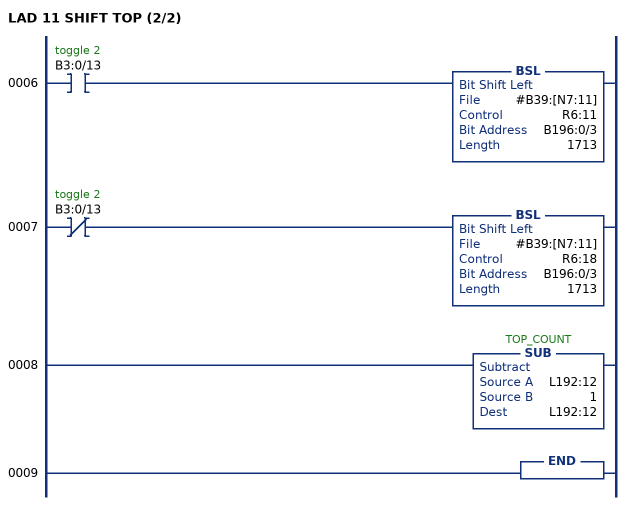
% Rung: 6 %
SOR XIC B3:0/13 BSL #B39:[N7:11] R6:11 B196:0/3 1713 EOR
%   B3:0/13  "toggle 2" %
%   N7:11  TOP_GOOD2_START_WORD %
%   B196:0/3  OFF %
% Rung: 7 %
SOR XIO B3:0/13 BSL #B39:[N7:11] R6:18 B196:0/3 1713 EOR
%   B3:0/13  "toggle 2" %
%   N7:11  TOP_GOOD2_START_WORD %
%   B196:0/3  OFF %
% Rung: 8 %
SOR SUB L192:12 1 L192:12 EOR
%   L192:12  TOP_COUNT %
% Rung: 9 %
SOR END EOR

LADDER 12 "BOTOPTIC"
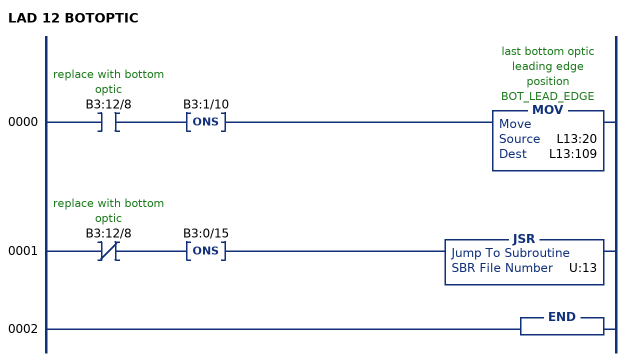
% Rung: 0 %
SOR XIC B3:12/8 ONS B3:1/10 MOV L13:20 L13:109 EOR
%   B3:12/8  "replace with bottom optic" %
%   L13:20  BOT_POSITION %
%   L13:109  BOT_LEAD_EDGE  "last bottom optic leading edge position" %
% Rung: 1 %
SOR XIO B3:12/8 ONS B3:0/15 JSR U:13 EOR
%   B3:12/8  "replace with bottom optic" %
% Rung: 2 %
SOR END EOR

LADDER 13 "BOTOPTMES"
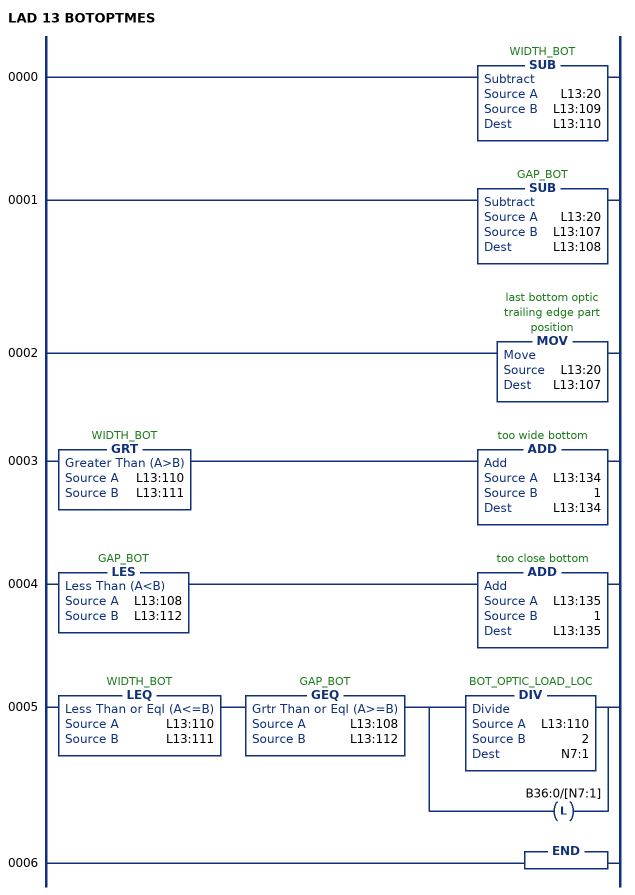
% Rung: 0 %
SOR SUB L13:20 L13:109 L13:110 EOR
%   L13:20  BOT_POSITION %
%   L13:109  BOT_LEAD_EDGE  "last bottom optic leading edge position" %
%   L13:110  WIDTH_BOT %
% Rung: 1 %
SOR SUB L13:20 L13:107 L13:108 EOR
%   L13:20  BOT_POSITION %
%   L13:107  "last bottom optic trailing edge part position" %
%   L13:108  GAP_BOT %
% Rung: 2 %
SOR MOV L13:20 L13:107 EOR
%   L13:20  BOT_POSITION %
%   L13:107  "last bottom optic trailing edge part position" %
% Rung: 3 %
SOR GRT L13:110 L13:111 ADD L13:134 1 L13:134 EOR
%   L13:110  WIDTH_BOT %
%   L13:111  BOT_MAX_WIDTH %
%   L13:134  "too wide bottom" %
% Rung: 4 %
SOR LES L13:108 L13:112 ADD L13:135 1 L13:135 EOR
%   L13:108  GAP_BOT %
%   L13:112  BOT_MIN_GAP %
%   L13:135  "too close bottom" %
% Rung: 5 %
SOR LEQ L13:110 L13:111 GEQ L13:108 L13:112 BST DIV L13:110 2 N7:1 NXB OTL B36:0/[N7:1] BND EOR
%   L13:110  WIDTH_BOT %
%   L13:111  BOT_MAX_WIDTH %
%   L13:108  GAP_BOT %
%   L13:112  BOT_MIN_GAP %
%   N7:1  BOT_OPTIC_LOAD_LOC %
%   B36:0  BOT_GOOD %
% Rung: 6 %
SOR END EOR

LADDER 135 "XFER"
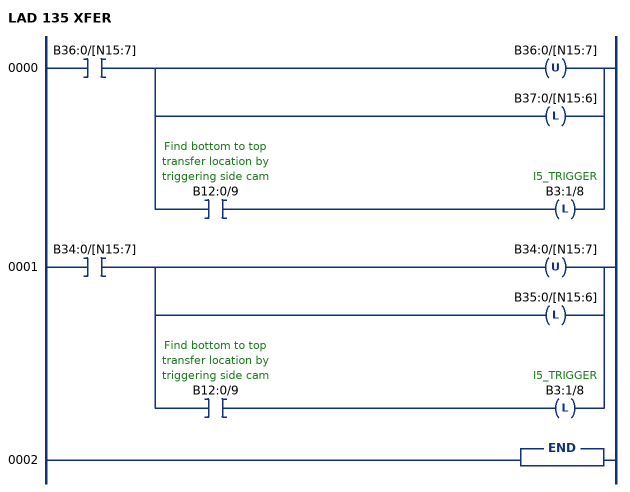
% Rung: 0 %
SOR XIC B36:0/[N15:7] BST OTU B36:0/[N15:7] NXB OTL B37:0/[N15:6] NXB XIC B12:0/9 OTL B3:1/8 BND EOR
%   B36:0  BOT_GOOD %
%   N15:7  XFER_OUT_LOC %
%   B37:0  TOPGOOD1 %
%   N15:6  XFER_IN_LOC %
%   B12:0/9  "Find bottom to top transfer location by triggering side cam" %
%   B3:1/8  I5_TRIGGER %
% Rung: 1 %
SOR XIC B34:0/[N15:7] BST OTU B34:0/[N15:7] NXB OTL B35:0/[N15:6] NXB XIC B12:0/9 OTL B3:1/8 BND EOR
%   B34:0  BOT_NG %
%   N15:7  XFER_OUT_LOC %
%   B35:0  TOP_NG %
%   N15:6  XFER_IN_LOC %
%   B12:0/9  "Find bottom to top transfer location by triggering side cam" %
%   B3:1/8  I5_TRIGGER %
% Rung: 2 %
SOR END EOR

LADDER 137 "TOPOPTIC"
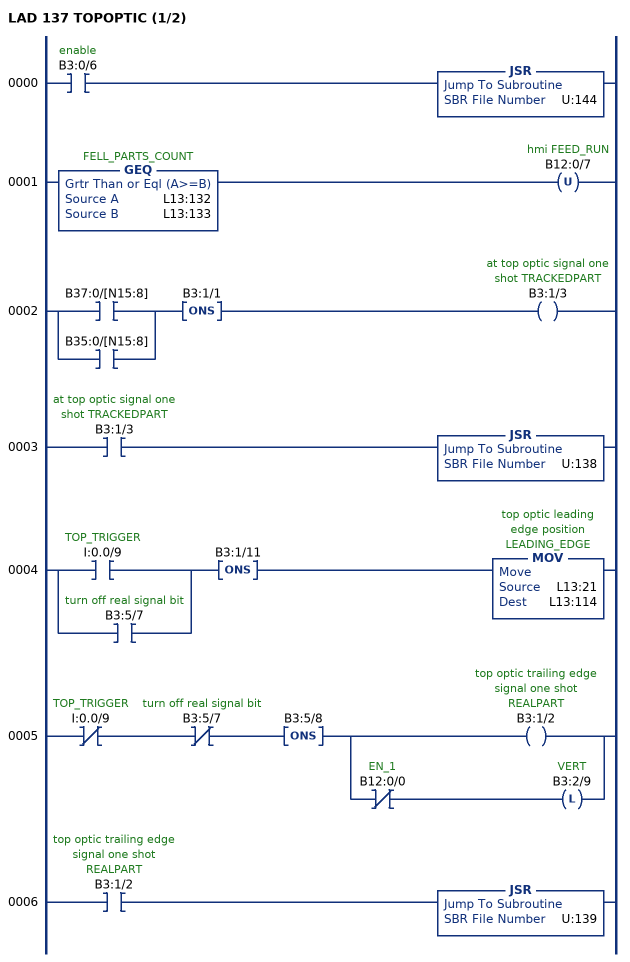
% Rung: 0 %
SOR XIC B3:0/6 JSR U:144 EOR
%   B3:0/6  "enable" %
% Rung: 1 %
SOR GEQ L13:132 L13:133 OTU B12:0/7 EOR
%   L13:132  FELL_PARTS_COUNT %
%   L13:133  FELL_PARTS_LIMIT %
%   B12:0/7  FEED_RUN  "hmi" %
% Rung: 2 %
SOR BST XIC B37:0/[N15:8] NXB XIC B35:0/[N15:8] BND ONS B3:1/1 OTE B3:1/3 EOR
%   B37:0  TOPGOOD1 %
%   N15:8  TOP_OPTIC_LOC %
%   B35:0  TOP_NG %
%   B3:1/3  TRACKEDPART  "at top optic signal one shot" %
% Rung: 3 %
SOR XIC B3:1/3 JSR U:138 EOR
%   B3:1/3  TRACKEDPART  "at top optic signal one shot" %
% Rung: 4 %
SOR BST XIC I:0.0/9 NXB XIC B3:5/7 BND ONS B3:1/11 MOV L13:21 L13:114 EOR
%   I:0.0/9  TOP_TRIGGER %
%   B3:5/7  "turn off real signal bit" %
%   L13:21  TOP_POSITION %
%   L13:114  LEADING_EDGE  "top optic leading edge position" %
% Rung: 5 %
SOR XIO I:0.0/9 XIO B3:5/7 ONS B3:5/8 BST OTE B3:1/2 NXB XIO B12:0/0 OTL B3:2/9 BND EOR
%   I:0.0/9  TOP_TRIGGER %
%   B3:5/7  "turn off real signal bit" %
%   B3:1/2  REALPART  "top optic trailing edge signal one shot" %
%   B12:0/0  EN_1 %
%   B3:2/9  VERT %
% Rung: 6 %
SOR XIC B3:1/2 JSR U:139 EOR
%   B3:1/2  REALPART  "top optic trailing edge signal one shot" %

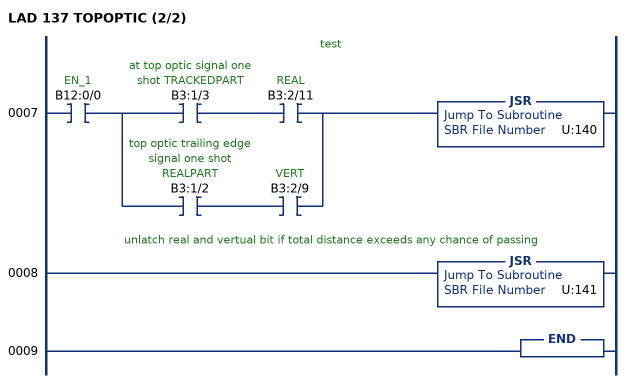
% Rung: 7 %
% test %
SOR XIC B12:0/0 BST XIC B3:1/3 XIC B3:2/11 NXB XIC B3:1/2 XIC B3:2/9 BND JSR U:140 EOR
%   B12:0/0  EN_1 %
%   B3:1/3  TRACKEDPART  "at top optic signal one shot" %
%   B3:2/11  REAL %
%   B3:1/2  REALPART  "top optic trailing edge signal one shot" %
%   B3:2/9  VERT %
% Rung: 8 %
% unlatch real and vertual bit if total distance exceeds any chance of passing %
SOR JSR U:141 EOR
% Rung: 9 %
SOR END EOR

LADDER 138 "TOPOPVERT"
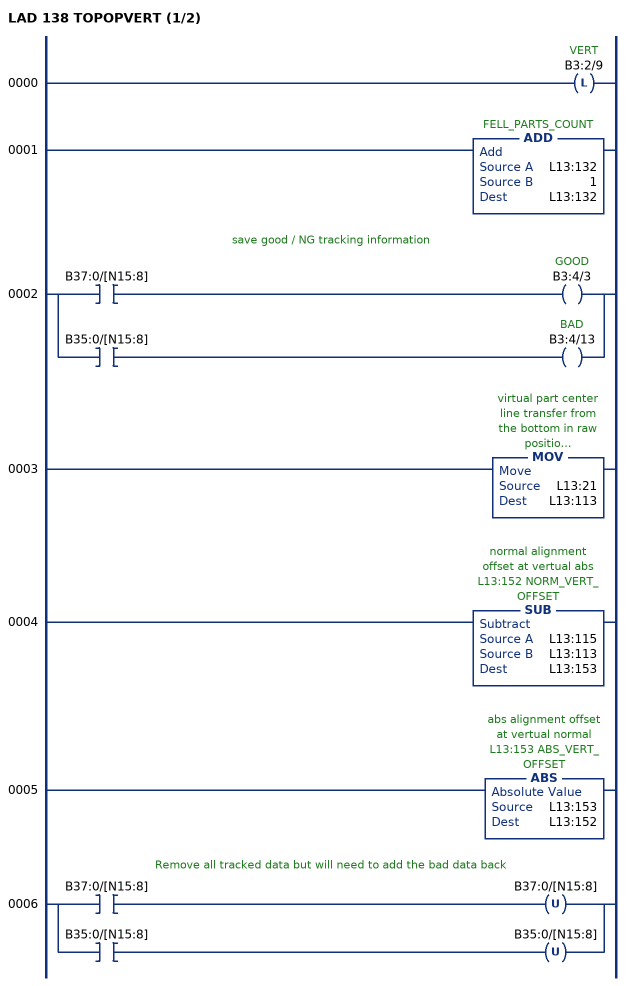
% Rung: 0 %
SOR OTL B3:2/9 EOR
%   B3:2/9  VERT %
% Rung: 1 %
SOR ADD L13:132 1 L13:132 EOR
%   L13:132  FELL_PARTS_COUNT %
% Rung: 2 %
% save good / NG tracking information %
SOR BST XIC B37:0/[N15:8] OTE B3:4/3 NXB XIC B35:0/[N15:8] OTE B3:4/13 BND EOR
%   B37:0  TOPGOOD1 %
%   N15:8  TOP_OPTIC_LOC %
%   B3:4/3  GOOD %
%   B35:0  TOP_NG %
%   B3:4/13  BAD %
% Rung: 3 %
SOR MOV L13:21 L13:113 EOR
%   L13:21  TOP_POSITION %
%   L13:113  VERTUAL_PT_RAW_CL  "virtual part center line transfer from the bottom in raw position" %
% Rung: 4 %
SOR SUB L13:115 L13:113 L13:153 EOR
%   L13:115  TRAILING_EDGE_RAW  "top optic trailing edge position" %
%   L13:113  VERTUAL_PT_RAW_CL  "virtual part center line transfer from the bottom in raw position" %
%   L13:153  NORM_VERT_OFFSET  "normal alignment offset at vertual abs L13:152" %
% Rung: 5 %
SOR ABS L13:153 L13:152 EOR
%   L13:153  NORM_VERT_OFFSET  "normal alignment offset at vertual abs L13:152" %
%   L13:152  ABS_VERT_OFFSET  "abs alignment offset at vertual normal L13:153" %
% Rung: 6 %
% Remove all tracked data but will need to add the bad data back %
SOR BST XIC B37:0/[N15:8] OTU B37:0/[N15:8] NXB XIC B35:0/[N15:8] OTU B35:0/[N15:8] BND EOR
%   B37:0  TOPGOOD1 %
%   N15:8  TOP_OPTIC_LOC %
%   B35:0  TOP_NG %

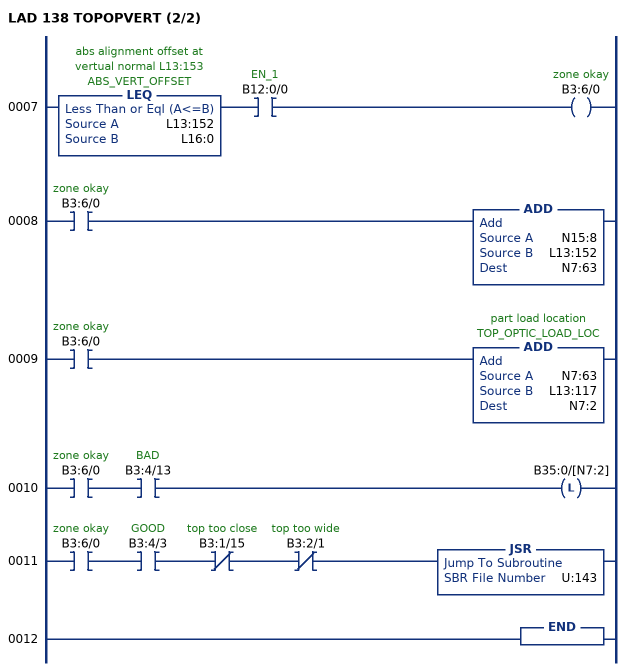
% Rung: 7 %
SOR LEQ L13:152 L16:0 XIC B12:0/0 OTE B3:6/0 EOR
%   L13:152  ABS_VERT_OFFSET  "abs alignment offset at vertual normal L13:153" %
%   L16:0  MAX_OFFSET %
%   B12:0/0  EN_1 %
%   B3:6/0  "zone okay" %
% Rung: 8 %
SOR XIC B3:6/0 ADD N15:8 L13:152 N7:63 EOR
%   B3:6/0  "zone okay" %
%   N15:8  TOP_OPTIC_LOC %
%   L13:152  ABS_VERT_OFFSET  "abs alignment offset at vertual normal L13:153" %
% Rung: 9 %
SOR XIC B3:6/0 ADD N7:63 L13:117 N7:2 EOR
%   B3:6/0  "zone okay" %
%   L13:117  HALF_WIDTH  "1/2 width top" %
%   N7:2  TOP_OPTIC_LOAD_LOC  "part load location" %
% Rung: 10 %
SOR XIC B3:6/0 XIC B3:4/13 OTL B35:0/[N7:2] EOR
%   B3:6/0  "zone okay" %
%   B3:4/13  BAD %
%   B35:0  TOP_NG %
%   N7:2  TOP_OPTIC_LOAD_LOC  "part load location" %
% Rung: 11 %
SOR XIC B3:6/0 XIC B3:4/3 XIO B3:1/15 XIO B3:2/1 JSR U:143 EOR
%   B3:6/0  "zone okay" %
%   B3:4/3  GOOD %
%   B3:1/15  "top too close" %
%   B3:2/1  "top too wide" %
% Rung: 12 %
SOR END EOR

LADDER 139 "TOPOPREAL"
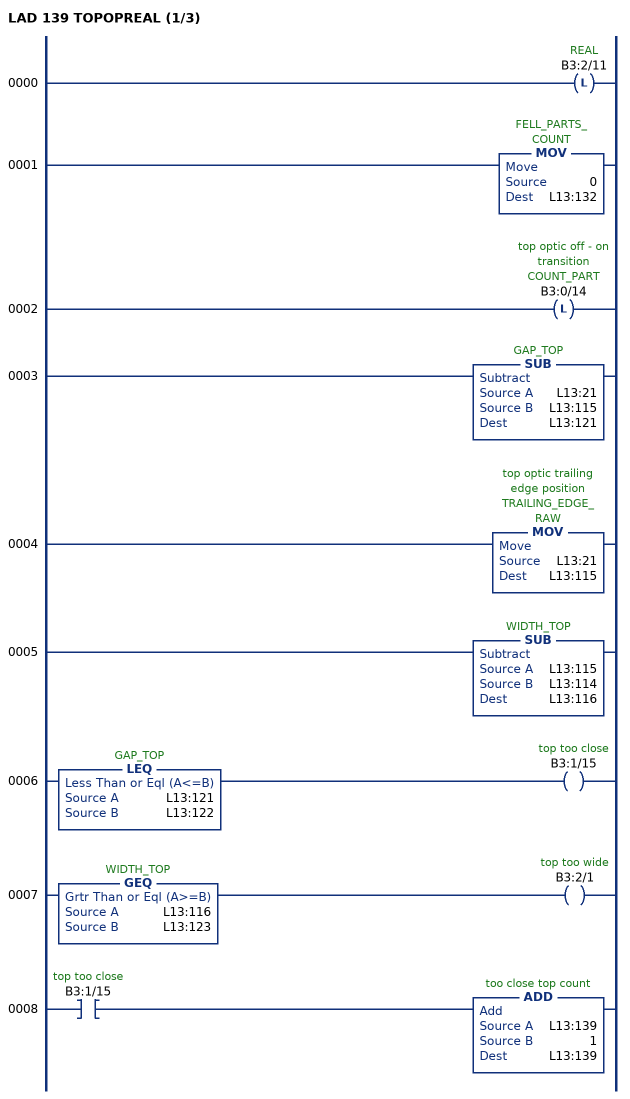
% Rung: 0 %
SOR OTL B3:2/11 EOR
%   B3:2/11  REAL %
% Rung: 1 %
SOR MOV 0 L13:132 EOR
%   L13:132  FELL_PARTS_COUNT %
% Rung: 2 %
SOR OTL B3:0/14 EOR
%   B3:0/14  COUNT_PART  "top optic off - on transition" %
% Rung: 3 %
SOR SUB L13:21 L13:115 L13:121 EOR
%   L13:21  TOP_POSITION %
%   L13:115  TRAILING_EDGE_RAW  "top optic trailing edge position" %
%   L13:121  GAP_TOP %
% Rung: 4 %
SOR MOV L13:21 L13:115 EOR
%   L13:21  TOP_POSITION %
%   L13:115  TRAILING_EDGE_RAW  "top optic trailing edge position" %
% Rung: 5 %
SOR SUB L13:115 L13:114 L13:116 EOR
%   L13:115  TRAILING_EDGE_RAW  "top optic trailing edge position" %
%   L13:114  LEADING_EDGE  "top optic leading edge position" %
%   L13:116  WIDTH_TOP %
% Rung: 6 %
SOR LEQ L13:121 L13:122 OTE B3:1/15 EOR
%   L13:121  GAP_TOP %
%   L13:122  MIN_GAP_TOP %
%   B3:1/15  "top too close" %
% Rung: 7 %
SOR GEQ L13:116 L13:123 OTE B3:2/1 EOR
%   L13:116  WIDTH_TOP %
%   L13:123  MAX_WIDTH_TOP %
%   B3:2/1  "top too wide" %
% Rung: 8 %
SOR XIC B3:1/15 ADD L13:139 1 L13:139 EOR
%   B3:1/15  "top too close" %
%   L13:139  "too close top count" %

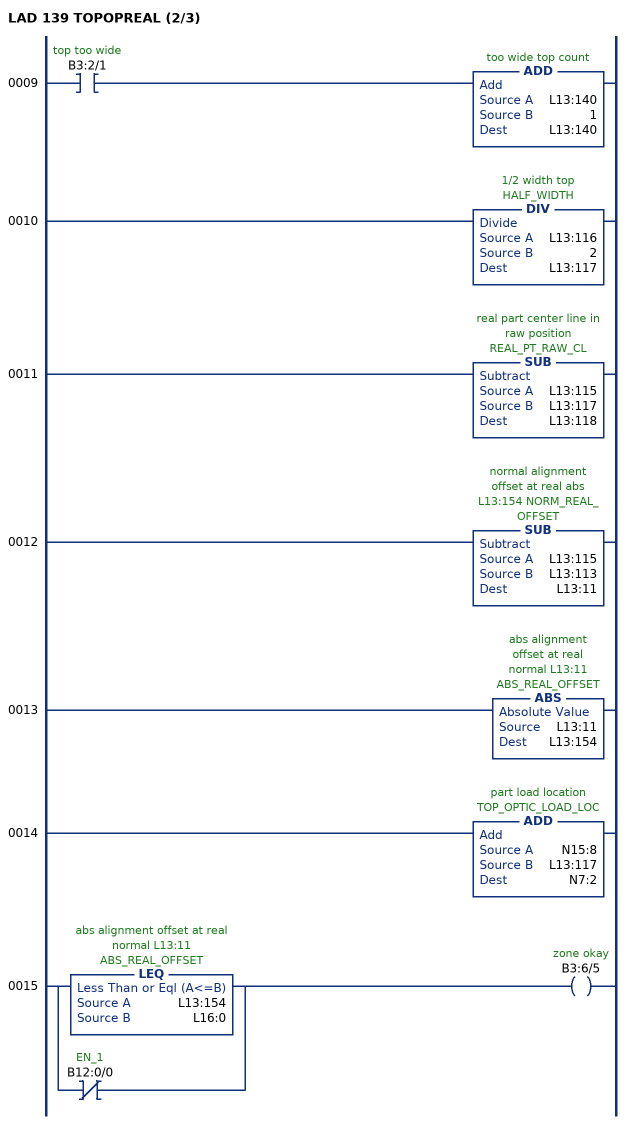
% Rung: 9 %
SOR XIC B3:2/1 ADD L13:140 1 L13:140 EOR
%   B3:2/1  "top too wide" %
%   L13:140  "too wide top count" %
% Rung: 10 %
SOR DIV L13:116 2 L13:117 EOR
%   L13:116  WIDTH_TOP %
%   L13:117  HALF_WIDTH  "1/2 width top" %
% Rung: 11 %
SOR SUB L13:115 L13:117 L13:118 EOR
%   L13:115  TRAILING_EDGE_RAW  "top optic trailing edge position" %
%   L13:117  HALF_WIDTH  "1/2 width top" %
%   L13:118  REAL_PT_RAW_CL  "real part center line in raw position" %
% Rung: 12 %
SOR SUB L13:115 L13:113 L13:11 EOR
%   L13:115  TRAILING_EDGE_RAW  "top optic trailing edge position" %
%   L13:113  VERTUAL_PT_RAW_CL  "virtual part center line transfer from the bottom in raw position" %
%   L13:11  NORM_REAL_OFFSET  "normal alignment offset at real abs L13:154" %
% Rung: 13 %
SOR ABS L13:11 L13:154 EOR
%   L13:11  NORM_REAL_OFFSET  "normal alignment offset at real abs L13:154" %
%   L13:154  ABS_REAL_OFFSET  "abs alignment offset at real normal L13:11" %
% Rung: 14 %
SOR ADD N15:8 L13:117 N7:2 EOR
%   N15:8  TOP_OPTIC_LOC %
%   L13:117  HALF_WIDTH  "1/2 width top" %
%   N7:2  TOP_OPTIC_LOAD_LOC  "part load location" %
% Rung: 15 %
SOR BST LEQ L13:154 L16:0 NXB XIO B12:0/0 BND OTE B3:6/5 EOR
%   L13:154  ABS_REAL_OFFSET  "abs alignment offset at real normal L13:11" %
%   L16:0  MAX_OFFSET %
%   B12:0/0  EN_1 %
%   B3:6/5  "zone okay" %

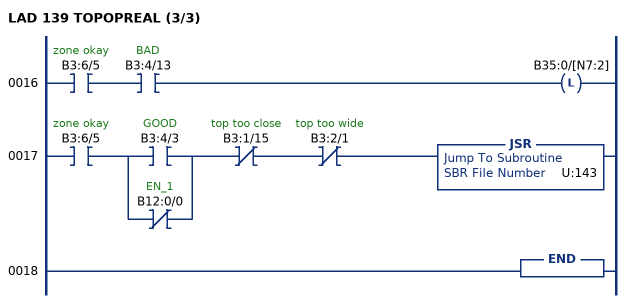
% Rung: 16 %
SOR XIC B3:6/5 XIC B3:4/13 OTL B35:0/[N7:2] EOR
%   B3:6/5  "zone okay" %
%   B3:4/13  BAD %
%   B35:0  TOP_NG %
%   N7:2  TOP_OPTIC_LOAD_LOC  "part load location" %
% Rung: 17 %
SOR XIC B3:6/5 BST XIC B3:4/3 NXB XIO B12:0/0 BND XIO B3:1/15 XIO B3:2/1 JSR U:143 EOR
%   B3:6/5  "zone okay" %
%   B3:4/3  GOOD %
%   B12:0/0  EN_1 %
%   B3:1/15  "top too close" %
%   B3:2/1  "top too wide" %
% Rung: 18 %
SOR END EOR

LADDER 140 "TOPOPTEST"
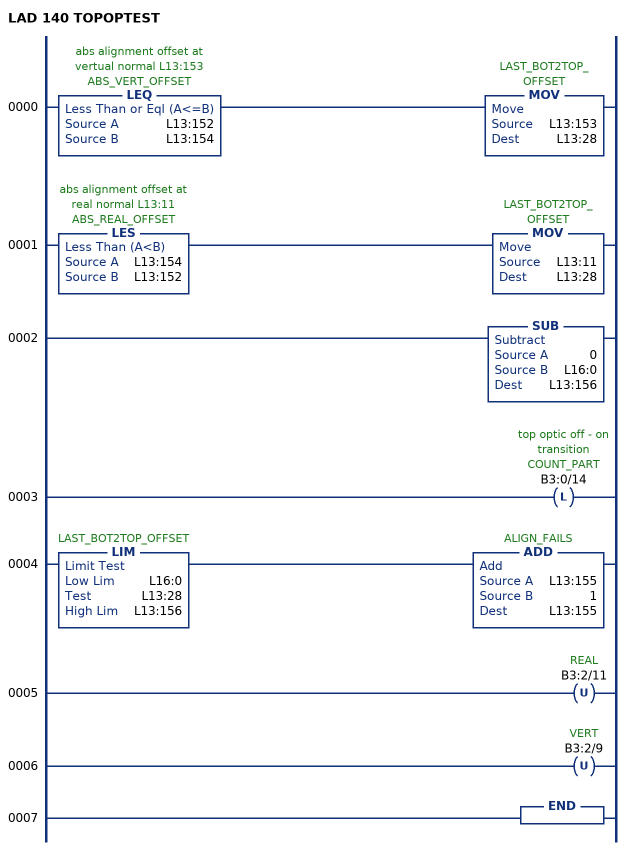
% Rung: 0 %
SOR LEQ L13:152 L13:154 MOV L13:153 L13:28 EOR
%   L13:152  ABS_VERT_OFFSET  "abs alignment offset at vertual normal L13:153" %
%   L13:154  ABS_REAL_OFFSET  "abs alignment offset at real normal L13:11" %
%   L13:153  NORM_VERT_OFFSET  "normal alignment offset at vertual abs L13:152" %
%   L13:28  LAST_BOT2TOP_OFFSET %
% Rung: 1 %
SOR LES L13:154 L13:152 MOV L13:11 L13:28 EOR
%   L13:154  ABS_REAL_OFFSET  "abs alignment offset at real normal L13:11" %
%   L13:152  ABS_VERT_OFFSET  "abs alignment offset at vertual normal L13:153" %
%   L13:11  NORM_REAL_OFFSET  "normal alignment offset at real abs L13:154" %
%   L13:28  LAST_BOT2TOP_OFFSET %
% Rung: 2 %
SOR SUB 0 L16:0 L13:156 EOR
%   L16:0  MAX_OFFSET %
% Rung: 3 %
SOR OTL B3:0/14 EOR
%   B3:0/14  COUNT_PART  "top optic off - on transition" %
% Rung: 4 %
SOR LIM L16:0 L13:28 L13:156 ADD L13:155 1 L13:155 EOR
%   L16:0  MAX_OFFSET %
%   L13:28  LAST_BOT2TOP_OFFSET %
%   L13:155  ALIGN_FAILS %
% Rung: 5 %
SOR OTU B3:2/11 EOR
%   B3:2/11  REAL %
% Rung: 6 %
SOR OTU B3:2/9 EOR
%   B3:2/9  VERT %
% Rung: 7 %
SOR END EOR

LADDER 141 "TOPOPRANGE"
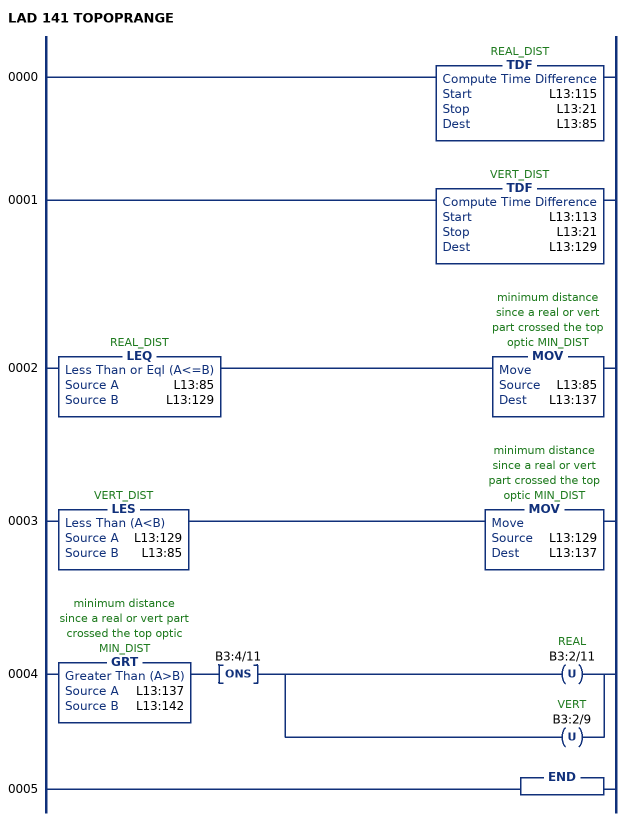
% Rung: 0 %
SOR TDF L13:115 L13:21 L13:85 EOR
%   L13:115  TRAILING_EDGE_RAW  "top optic trailing edge position" %
%   L13:21  TOP_POSITION %
%   L13:85  REAL_DIST %
% Rung: 1 %
SOR TDF L13:113 L13:21 L13:129 EOR
%   L13:113  VERTUAL_PT_RAW_CL  "virtual part center line transfer from the bottom in raw position" %
%   L13:21  TOP_POSITION %
%   L13:129  VERT_DIST %
% Rung: 2 %
SOR LEQ L13:85 L13:129 MOV L13:85 L13:137 EOR
%   L13:85  REAL_DIST %
%   L13:129  VERT_DIST %
%   L13:137  MIN_DIST  "minimum distance since a real or vert part crossed the top optic" %
% Rung: 3 %
SOR LES L13:129 L13:85 MOV L13:129 L13:137 EOR
%   L13:129  VERT_DIST %
%   L13:85  REAL_DIST %
%   L13:137  MIN_DIST  "minimum distance since a real or vert part crossed the top optic" %
% Rung: 4 %
SOR GRT L13:137 L13:142 ONS B3:4/11 BST OTU B3:2/11 NXB OTU B3:2/9 BND EOR
%   L13:137  MIN_DIST  "minimum distance since a real or vert part crossed the top optic" %
%   L13:142  LAST_ALIGNMENT_FAILS %
%   B3:2/11  REAL %
%   B3:2/9  VERT %
% Rung: 5 %
SOR END EOR

LADDER 142 "TOPOPRANGE"
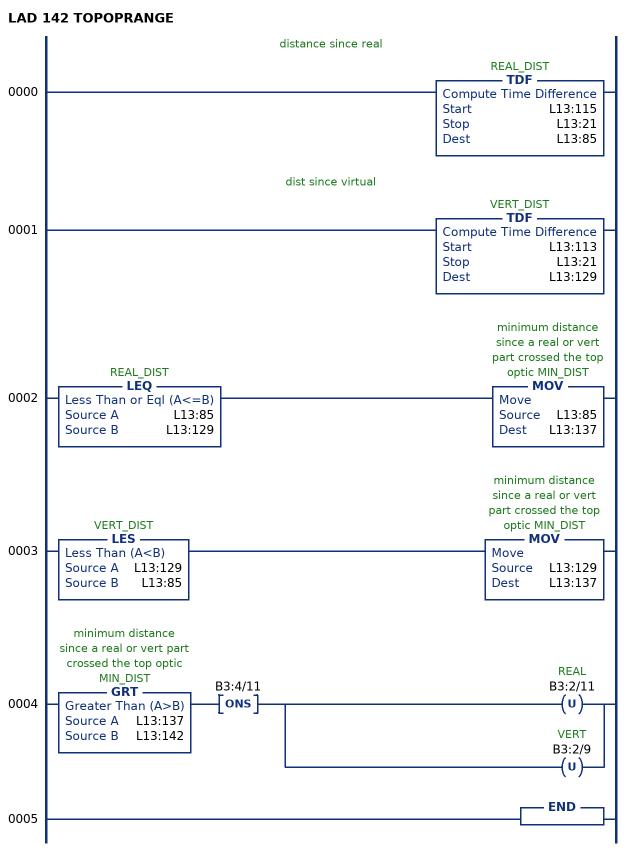
% Rung: 0 %
% distance since real %
SOR TDF L13:115 L13:21 L13:85 EOR
%   L13:115  TRAILING_EDGE_RAW  "top optic trailing edge position" %
%   L13:21  TOP_POSITION %
%   L13:85  REAL_DIST %
% Rung: 1 %
% dist since virtual %
SOR TDF L13:113 L13:21 L13:129 EOR
%   L13:113  VERTUAL_PT_RAW_CL  "virtual part center line transfer from the bottom in raw position" %
%   L13:21  TOP_POSITION %
%   L13:129  VERT_DIST %
% Rung: 2 %
SOR LEQ L13:85 L13:129 MOV L13:85 L13:137 EOR
%   L13:85  REAL_DIST %
%   L13:129  VERT_DIST %
%   L13:137  MIN_DIST  "minimum distance since a real or vert part crossed the top optic" %
% Rung: 3 %
SOR LES L13:129 L13:85 MOV L13:129 L13:137 EOR
%   L13:129  VERT_DIST %
%   L13:85  REAL_DIST %
%   L13:137  MIN_DIST  "minimum distance since a real or vert part crossed the top optic" %
% Rung: 4 %
SOR GRT L13:137 L13:142 ONS B3:4/11 BST OTU B3:2/11 NXB OTU B3:2/9 BND EOR
%   L13:137  MIN_DIST  "minimum distance since a real or vert part crossed the top optic" %
%   L13:142  LAST_ALIGNMENT_FAILS %
%   B3:2/11  REAL %
%   B3:2/9  VERT %
% Rung: 5 %
SOR END EOR

LADDER 143 "TOPOPOKAY"
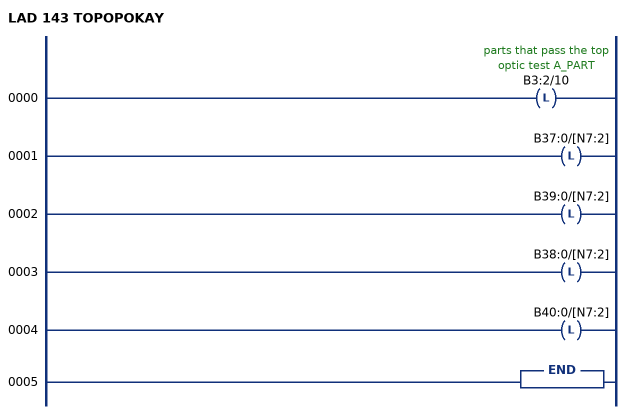
% Rung: 0 %
SOR OTL B3:2/10 EOR
%   B3:2/10  A_PART  "parts that pass the top optic test" %
% Rung: 1 %
SOR OTL B37:0/[N7:2] EOR
%   B37:0  TOPGOOD1 %
%   N7:2  TOP_OPTIC_LOAD_LOC  "part load location" %
% Rung: 2 %
SOR OTL B39:0/[N7:2] EOR
%   B39:0  TOPGOOD2 %
%   N7:2  TOP_OPTIC_LOAD_LOC  "part load location" %
% Rung: 3 %
SOR OTL B38:0/[N7:2] EOR
%   B38:0  EX1_GOOD %
%   N7:2  TOP_OPTIC_LOAD_LOC  "part load location" %
% Rung: 4 %
SOR OTL B40:0/[N7:2] EOR
%   B40:0  EX3_GOOD %
%   N7:2  TOP_OPTIC_LOAD_LOC  "part load location" %
% Rung: 5 %
SOR END EOR

LADDER 144 "TESTINJECT"
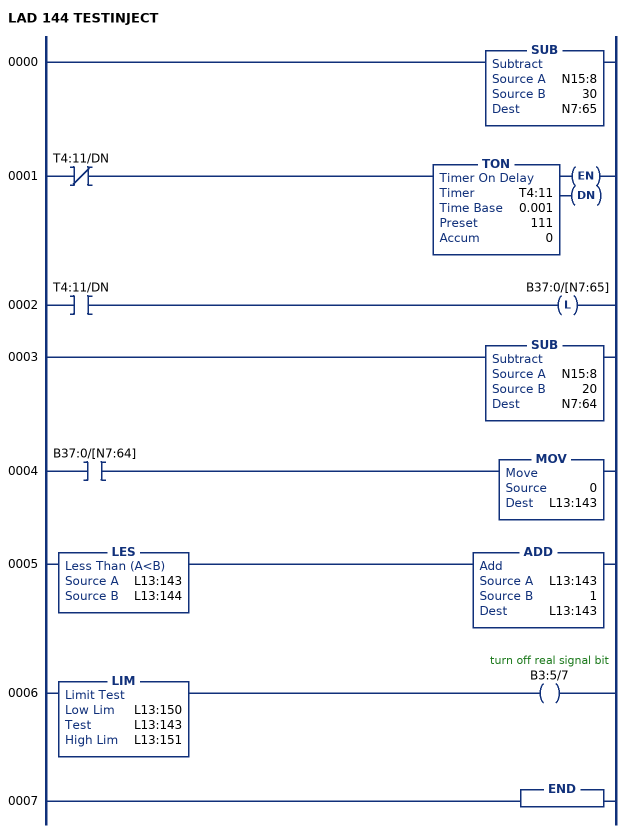
% Rung: 0 %
SOR SUB N15:8 30 N7:65 EOR
%   N15:8  TOP_OPTIC_LOC %
% Rung: 1 %
SOR XIO T4:11/DN TON T4:11 0.001 111 0 EOR
% Rung: 2 %
SOR XIC T4:11/DN OTL B37:0/[N7:65] EOR
%   B37:0  TOPGOOD1 %
% Rung: 3 %
SOR SUB N15:8 20 N7:64 EOR
%   N15:8  TOP_OPTIC_LOC %
% Rung: 4 %
SOR XIC B37:0/[N7:64] MOV 0 L13:143 EOR
%   B37:0  TOPGOOD1 %
% Rung: 5 %
SOR LES L13:143 L13:144 ADD L13:143 1 L13:143 EOR
% Rung: 6 %
SOR LIM L13:150 L13:143 L13:151 OTE B3:5/7 EOR
%   B3:5/7  "turn off real signal bit" %
% Rung: 7 %
SOR END EOR

LADDER 148 "I5"
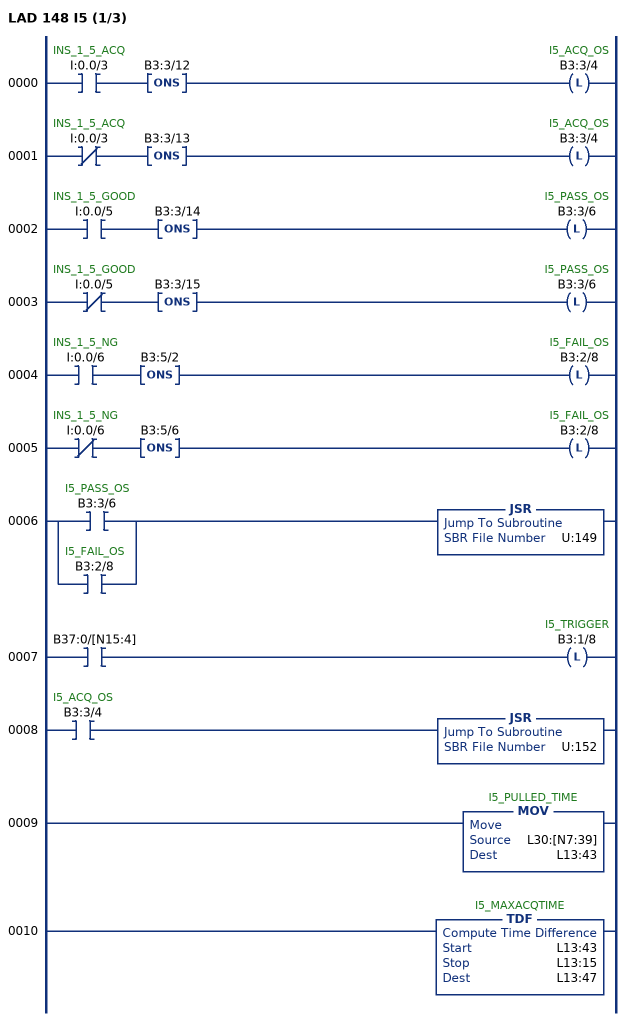
% Rung: 0 %
SOR XIC I:0.0/3 ONS B3:3/12 OTL B3:3/4 EOR
%   I:0.0/3  INS_1_5_ACQ %
%   B3:3/4  I5_ACQ_OS %
% Rung: 1 %
SOR XIO I:0.0/3 ONS B3:3/13 OTL B3:3/4 EOR
%   I:0.0/3  INS_1_5_ACQ %
%   B3:3/4  I5_ACQ_OS %
% Rung: 2 %
SOR XIC I:0.0/5 ONS B3:3/14 OTL B3:3/6 EOR
%   I:0.0/5  INS_1_5_GOOD %
%   B3:3/6  I5_PASS_OS %
% Rung: 3 %
SOR XIO I:0.0/5 ONS B3:3/15 OTL B3:3/6 EOR
%   I:0.0/5  INS_1_5_GOOD %
%   B3:3/6  I5_PASS_OS %
% Rung: 4 %
SOR XIC I:0.0/6 ONS B3:5/2 OTL B3:2/8 EOR
%   I:0.0/6  INS_1_5_NG %
%   B3:2/8  I5_FAIL_OS %
% Rung: 5 %
SOR XIO I:0.0/6 ONS B3:5/6 OTL B3:2/8 EOR
%   I:0.0/6  INS_1_5_NG %
%   B3:2/8  I5_FAIL_OS %
% Rung: 6 %
SOR BST XIC B3:3/6 NXB XIC B3:2/8 BND JSR U:149 EOR
%   B3:3/6  I5_PASS_OS %
%   B3:2/8  I5_FAIL_OS %
% Rung: 7 %
SOR XIC B37:0/[N15:4] OTL B3:1/8 EOR
%   B37:0  TOPGOOD1 %
%   N15:4  I5_TRIG_LOC %
%   B3:1/8  I5_TRIGGER %
% Rung: 8 %
SOR XIC B3:3/4 JSR U:152 EOR
%   B3:3/4  I5_ACQ_OS %
% Rung: 9 %
SOR MOV L30:[N7:39] L13:43 EOR
%   N7:39  I5_OLDEST_PART_INDEX %
%   L13:43  I5_PULLED_TIME %
% Rung: 10 %
SOR TDF L13:43 L13:15 L13:47 EOR
%   L13:43  I5_PULLED_TIME %
%   L13:15  THE_TIME %
%   L13:47  I5_MAXACQTIME %

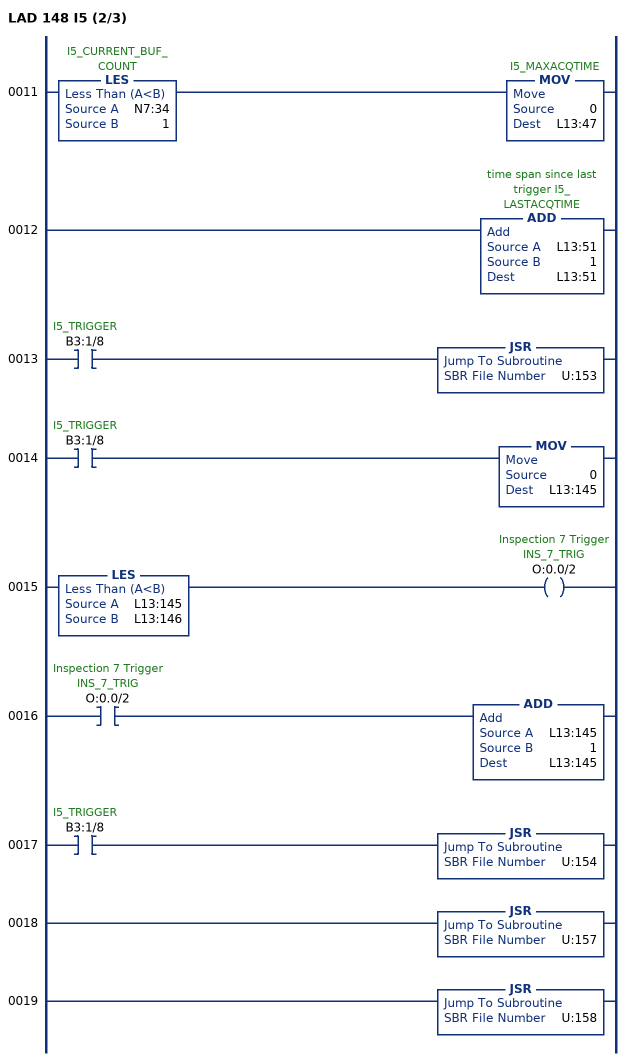
% Rung: 11 %
SOR LES N7:34 1 MOV 0 L13:47 EOR
%   N7:34  I5_CURRENT_BUF_COUNT %
%   L13:47  I5_MAXACQTIME %
% Rung: 12 %
SOR ADD L13:51 1 L13:51 EOR
%   L13:51  I5_LASTACQTIME  "time span since last trigger" %
% Rung: 13 %
SOR XIC B3:1/8 JSR U:153 EOR
%   B3:1/8  I5_TRIGGER %
% Rung: 14 %
SOR XIC B3:1/8 MOV 0 L13:145 EOR
%   B3:1/8  I5_TRIGGER %
% Rung: 15 %
SOR LES L13:145 L13:146 OTE O:0.0/2 EOR
%   O:0.0/2  INS_7_TRIG  "Inspection 7 Trigger" %
% Rung: 16 %
SOR XIC O:0.0/2 ADD L13:145 1 L13:145 EOR
%   O:0.0/2  INS_7_TRIG  "Inspection 7 Trigger" %
% Rung: 17 %
SOR XIC B3:1/8 JSR U:154 EOR
%   B3:1/8  I5_TRIGGER %
% Rung: 18 %
SOR JSR U:157 EOR
% Rung: 19 %
SOR JSR U:158 EOR

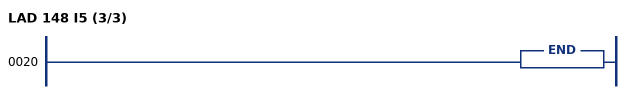
% Rung: 20 %
SOR END EOR

LADDER 149 "I5 RESULT"
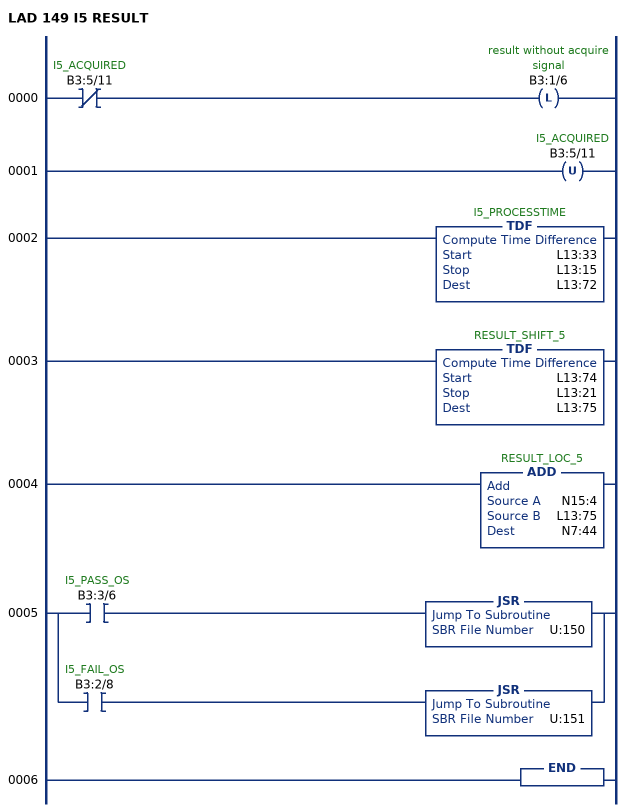
% Rung: 0 %
SOR XIO B3:5/11 OTL B3:1/6 EOR
%   B3:5/11  I5_ACQUIRED %
%   B3:1/6  "result without acquire signal" %
% Rung: 1 %
SOR OTU B3:5/11 EOR
%   B3:5/11  I5_ACQUIRED %
% Rung: 2 %
SOR TDF L13:33 L13:15 L13:72 EOR
%   L13:33  I5_TIMEOFACQ %
%   L13:15  THE_TIME %
%   L13:72  I5_PROCESSTIME %
% Rung: 3 %
SOR TDF L13:74 L13:21 L13:75 EOR
%   L13:74  I5_PROCESS_START_POS %
%   L13:21  TOP_POSITION %
%   L13:75  RESULT_SHIFT_5 %
% Rung: 4 %
SOR ADD N15:4 L13:75 N7:44 EOR
%   N15:4  I5_TRIG_LOC %
%   L13:75  RESULT_SHIFT_5 %
%   N7:44  RESULT_LOC_5 %
% Rung: 5 %
SOR BST XIC B3:3/6 JSR U:150 NXB XIC B3:2/8 JSR U:151 BND EOR
%   B3:3/6  I5_PASS_OS %
%   B3:2/8  I5_FAIL_OS %
% Rung: 6 %
SOR END EOR

LADDER 150 "I5 PASS"
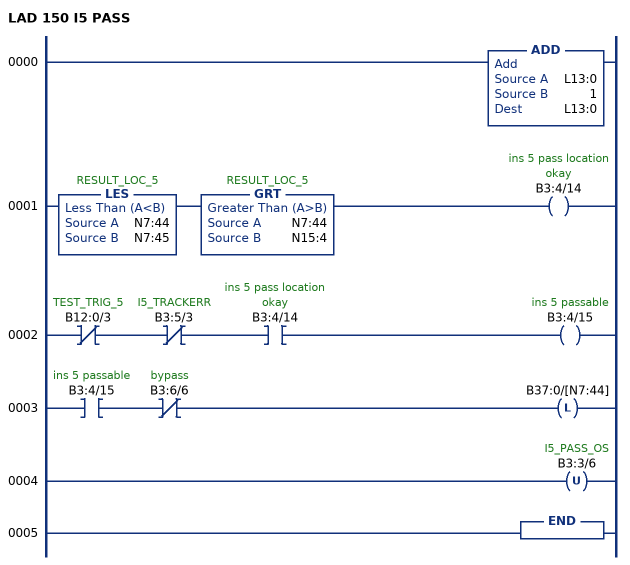
% Rung: 0 %
SOR ADD L13:0 1 L13:0 EOR
% Rung: 1 %
SOR LES N7:44 N7:45 GRT N7:44 N15:4 OTE B3:4/14 EOR
%   N7:44  RESULT_LOC_5 %
%   N7:45  I5_MAX_SHIFT  "ins 5 maximum result location" %
%   N15:4  I5_TRIG_LOC %
%   B3:4/14  "ins 5 pass location okay" %
% Rung: 2 %
SOR XIO B12:0/3 XIO B3:5/3 XIC B3:4/14 OTE B3:4/15 EOR
%   B12:0/3  TEST_TRIG_5 %
%   B3:5/3  I5_TRACKERR %
%   B3:4/14  "ins 5 pass location okay" %
%   B3:4/15  "ins 5 passable" %
% Rung: 3 %
SOR XIC B3:4/15 XIO B3:6/6 OTL B37:0/[N7:44] EOR
%   B3:4/15  "ins 5 passable" %
%   B3:6/6  "bypass" %
%   B37:0  TOPGOOD1 %
%   N7:44  RESULT_LOC_5 %
% Rung: 4 %
SOR OTU B3:3/6 EOR
%   B3:3/6  I5_PASS_OS %
% Rung: 5 %
SOR END EOR

LADDER 151 "I5 FAIL"
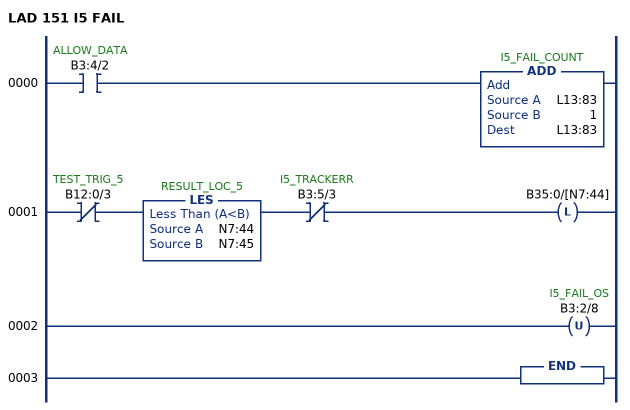
% Rung: 0 %
SOR XIC B3:4/2 ADD L13:83 1 L13:83 EOR
%   B3:4/2  ALLOW_DATA %
%   L13:83  I5_FAIL_COUNT %
% Rung: 1 %
SOR XIO B12:0/3 LES N7:44 N7:45 XIO B3:5/3 OTL B35:0/[N7:44] EOR
%   B12:0/3  TEST_TRIG_5 %
%   N7:44  RESULT_LOC_5 %
%   N7:45  I5_MAX_SHIFT  "ins 5 maximum result location" %
%   B3:5/3  I5_TRACKERR %
%   B35:0  TOP_NG %
% Rung: 2 %
SOR OTU B3:2/8 EOR
%   B3:2/8  I5_FAIL_OS %
% Rung: 3 %
SOR END EOR

LADDER 152 "I5 ACQ"
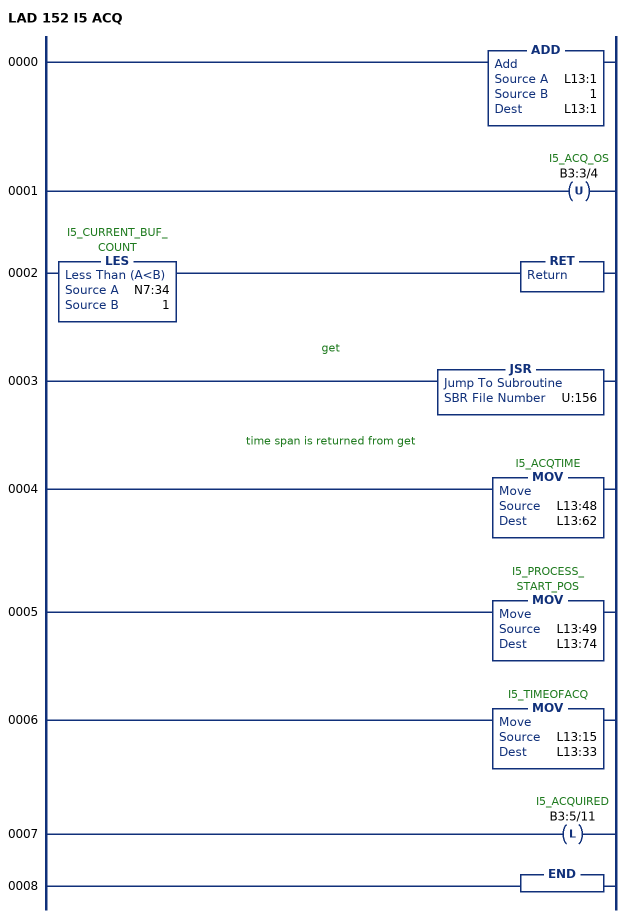
% Rung: 0 %
SOR ADD L13:1 1 L13:1 EOR
% Rung: 1 %
SOR OTU B3:3/4 EOR
%   B3:3/4  I5_ACQ_OS %
% Rung: 2 %
SOR LES N7:34 1 RET EOR
%   N7:34  I5_CURRENT_BUF_COUNT %
% Rung: 3 %
% get %
SOR JSR U:156 EOR
% Rung: 4 %
% time span is returned from get %
SOR MOV L13:48 L13:62 EOR
%   L13:48  I5_TIME_SPAN %
%   L13:62  I5_ACQTIME %
% Rung: 5 %
SOR MOV L13:49 L13:74 EOR
%   L13:49  I5_PULLED_POSITION %
%   L13:74  I5_PROCESS_START_POS %
% Rung: 6 %
SOR MOV L13:15 L13:33 EOR
%   L13:15  THE_TIME %
%   L13:33  I5_TIMEOFACQ %
% Rung: 7 %
SOR OTL B3:5/11 EOR
%   B3:5/11  I5_ACQUIRED %
% Rung: 8 %
SOR END EOR

LADDER 153 "I5 TESTER"
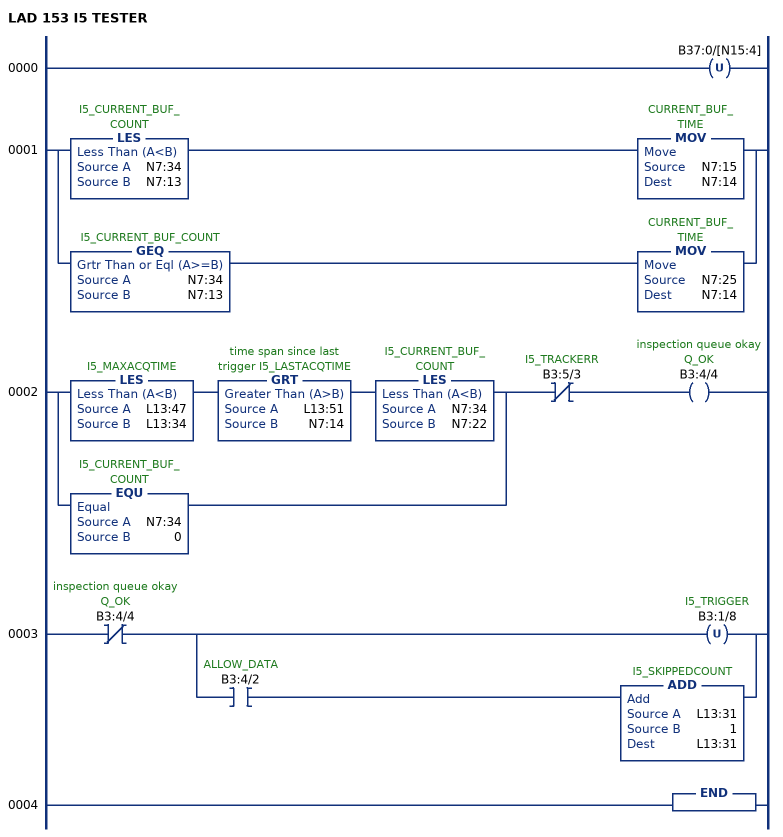
% Rung: 0 %
SOR OTU B37:0/[N15:4] EOR
%   B37:0  TOPGOOD1 %
%   N15:4  I5_TRIG_LOC %
% Rung: 1 %
SOR BST LES N7:34 N7:13 MOV N7:15 N7:14 NXB GEQ N7:34 N7:13 MOV N7:25 N7:14 BND EOR
%   N7:34  I5_CURRENT_BUF_COUNT %
%   N7:13  BUF_TRANS  "cam to pc buf transition" %
%   N7:15  CAM_BUF_TIME  "cam buf time" %
%   N7:14  CURRENT_BUF_TIME %
%   N7:25  PC_BUF_TIME  "pc buf time" %
% Rung: 2 %
SOR BST LES L13:47 L13:34 GRT L13:51 N7:14 LES N7:34 N7:22 NXB EQU N7:34 0 BND XIO B3:5/3 OTE B3:4/4 EOR
%   L13:47  I5_MAXACQTIME %
%   L13:34  MAX_ACQ_ALL  "absolute max acquire time before bypass trigger" %
%   L13:51  I5_LASTACQTIME  "time span since last trigger" %
%   N7:14  CURRENT_BUF_TIME %
%   N7:34  I5_CURRENT_BUF_COUNT %
%   N7:22  MAX_BUF_ALL  "max buffer count alowed before bypass" %
%   B3:5/3  I5_TRACKERR %
%   B3:4/4  Q_OK  "inspection queue okay" %
% Rung: 3 %
SOR XIO B3:4/4 BST OTU B3:1/8 NXB XIC B3:4/2 ADD L13:31 1 L13:31 BND EOR
%   B3:4/4  Q_OK  "inspection queue okay" %
%   B3:1/8  I5_TRIGGER %
%   B3:4/2  ALLOW_DATA %
%   L13:31  I5_SKIPPEDCOUNT %
% Rung: 4 %
SOR END EOR

LADDER 154 "I5 TRIG"
